FUNCTION Convert_TIME_TO_LINT : BOOL
VAR_INPUT
	in : TIME;
	out : REFERENCE TO LINT;
END_VAR
VAR
	converted : LINT;
END_VAR

converted := TIME_TO_LINT(in);

IF (LINT_TO_TIME(converted) <> in) THEN
	RETURN;
END_IF

out := converted;
Convert_TIME_TO_LINT := TRUE;

END_FUNCTION

(* stored: Version 1.1.0.1, ProductVersion 3.1.4024.12
   POU Convert_TIME_TO_LINT: Id {623764f2-0fff-4277-942b-10b880929160}, SpecialFunc None *)
